FUNCTION_BLOCK FB_GripperAction
VAR_INPUT
    bExecute       : BOOL;
    eCommand       : E_GripperCommand;
    bCancel        : BOOL;
    bAllowCloseTargetWithoutGrip : BOOL := FALSE;
    tAcceptTimeout : TIME := GVL_ProcessConfig.stGripper.tAcceptTimeout;
    tResultTimeout : TIME := GVL_ProcessConfig.stGripper.tResultTimeout;
END_VAR
VAR_IN_OUT
    ioGripper : ST_GripperInterface;
END_VAR
VAR_OUTPUT
    bBusy       : BOOL;
    bDone       : BOOL;
    bCloseTargetReachedWithoutGrip : BOOL;
    bError      : BOOL;
    udErrorCode : UDINT;
    udiActionId : UDINT;
    eStep       : E_GripperActionStep := E_GripperActionStep.Idle;
END_VAR
VAR
    bInitialized     : BOOL;
    bExecutePrevious : BOOL;
    eActiveCommand   : E_GripperCommand;
    bActiveAllowCloseTargetWithoutGrip : BOOL;
    fbAcceptTimeout  : TON;
    fbResultTimeout  : TON;
END_VAR

// 自动动作只写AutoCmd；底层Cmd由FB_GripperManager唯一生成。
IF NOT bInitialized THEN
    bExecutePrevious := bExecute;
    bInitialized := TRUE;
END_IF;

// 取消/释放只撤销特殊完成授权，不改变既有Stop/Fault链。
IF bCancel OR NOT bExecute THEN
    ioGripper.AutoCmd.bAllowCloseTargetWithoutGrip := FALSE;
    bActiveAllowCloseTargetWithoutGrip := FALSE;
    bCloseTargetReachedWithoutGrip := FALSE;
END_IF;

fbAcceptTimeout(
    IN := (eStep = E_GripperActionStep.WaitAccepted),
    PT := tAcceptTimeout
);
fbResultTimeout(
    IN := (eStep = E_GripperActionStep.WaitCompleted),
    PT := tResultTimeout
);

IF ((eStep = E_GripperActionStep.WaitAccepted)
    OR (eStep = E_GripperActionStep.WaitCompleted))
    AND (bCancel OR NOT bExecute) THEN
    bBusy := FALSE;
    bDone := FALSE;
    bError := TRUE;
    udErrorCode := TO_UDINT(E_GripperErrorCode.ActionCancelled);
    eStep := E_GripperActionStep.Error;
    bExecutePrevious := bExecute;
    RETURN;
END_IF;

CASE eStep OF
    E_GripperActionStep.Idle:
        bBusy := FALSE;
        bDone := FALSE;
        bCloseTargetReachedWithoutGrip := FALSE;
        bActiveAllowCloseTargetWithoutGrip := FALSE;
        bError := FALSE;
        udErrorCode := TO_UDINT(E_GripperErrorCode.None);

        IF bExecute AND NOT bExecutePrevious AND NOT bCancel THEN
            IF (eCommand <> E_GripperCommand.Close)
                AND (eCommand <> E_GripperCommand.Open)
                AND (eCommand <> E_GripperCommand.Enable) THEN
                bError := TRUE;
                udErrorCode := TO_UDINT(E_GripperErrorCode.ActionInvalidCommand);
                eStep := E_GripperActionStep.Error;
            ELSE
                eActiveCommand := eCommand;
                bActiveAllowCloseTargetWithoutGrip :=
                    bAllowCloseTargetWithoutGrip
                    AND (eActiveCommand = E_GripperCommand.Close);
                ioGripper.AutoCmd.bAllowCloseTargetWithoutGrip :=
                    bActiveAllowCloseTargetWithoutGrip;
                ioGripper.AutoCmd.eCommand := eActiveCommand;
                IF ioGripper.AutoCmd.udiRequestId = 16#FFFFFFFF THEN
                    ioGripper.AutoCmd.udiRequestId := 1;
                ELSE
                    ioGripper.AutoCmd.udiRequestId :=
                        ioGripper.AutoCmd.udiRequestId + 1;
                END_IF;
                udiActionId := ioGripper.AutoCmd.udiRequestId;
                bBusy := TRUE;
                eStep := E_GripperActionStep.WaitAccepted;
            END_IF;
        END_IF;

    E_GripperActionStep.WaitAccepted:
        IF ioGripper.AutoFeedback.udiRejectedId = udiActionId THEN
            bBusy := FALSE;
            bError := TRUE;
            udErrorCode := ioGripper.AutoFeedback.udErrorCode;
            IF udErrorCode = TO_UDINT(E_GripperErrorCode.None) THEN
                udErrorCode := TO_UDINT(E_GripperErrorCode.ActionResultInvalid);
            END_IF;
            eStep := E_GripperActionStep.Error;
        ELSIF ioGripper.AutoFeedback.udiFailedId = udiActionId THEN
            bBusy := FALSE;
            bError := TRUE;
            udErrorCode := ioGripper.AutoFeedback.udErrorCode;
            IF udErrorCode = TO_UDINT(E_GripperErrorCode.None) THEN
                udErrorCode := TO_UDINT(E_GripperErrorCode.ActionResultInvalid);
            END_IF;
            eStep := E_GripperActionStep.Error;
        ELSIF ioGripper.AutoFeedback.udiAcceptedId = udiActionId THEN
            eStep := E_GripperActionStep.WaitCompleted;
        ELSIF fbAcceptTimeout.Q THEN
            bBusy := FALSE;
            bError := TRUE;
            udErrorCode := TO_UDINT(E_GripperErrorCode.ActionAcceptTimeout);
            eStep := E_GripperActionStep.Error;
        END_IF;

    E_GripperActionStep.WaitCompleted:
        IF ioGripper.AutoFeedback.udiFailedId = udiActionId THEN
            bBusy := FALSE;
            bError := TRUE;
            udErrorCode := ioGripper.AutoFeedback.udErrorCode;
            IF udErrorCode = TO_UDINT(E_GripperErrorCode.None) THEN
                udErrorCode := TO_UDINT(E_GripperErrorCode.ActionResultInvalid);
            END_IF;
            eStep := E_GripperActionStep.Error;
        ELSIF ioGripper.AutoFeedback.udiCompletedId = udiActionId THEN
            IF ioGripper.State.bHealthy
                AND ((eActiveCommand <> E_GripperCommand.Enable)
                    OR (ioGripper.AutoFeedback.udErrorCode = TO_UDINT(E_GripperErrorCode.None)))
                AND ((eActiveCommand = E_GripperCommand.Enable)
                    OR NOT ioGripper.AutoFeedback.bCloseTargetReachedWithoutGrip
                    OR bActiveAllowCloseTargetWithoutGrip) THEN
                bBusy := FALSE;
                bCloseTargetReachedWithoutGrip :=
                    ioGripper.AutoFeedback.bCloseTargetReachedWithoutGrip;
                bDone := TRUE;
                eStep := E_GripperActionStep.Done;
            ELSE
                bBusy := FALSE;
                bError := TRUE;
                udErrorCode := TO_UDINT(E_GripperErrorCode.ActionResultInvalid);
                eStep := E_GripperActionStep.Error;
            END_IF;
        ELSIF fbResultTimeout.Q THEN
            bBusy := FALSE;
            bError := TRUE;
            udErrorCode := TO_UDINT(E_GripperErrorCode.ActionResultTimeout);
            eStep := E_GripperActionStep.Error;
        END_IF;

    E_GripperActionStep.Done:
        bBusy := FALSE;
        IF NOT bExecute THEN
            bDone := FALSE;
            eStep := E_GripperActionStep.Idle;
        ELSIF NOT ioGripper.State.bHealthy
            OR (ioGripper.AutoFeedback.udiCompletedId <> udiActionId) THEN
            bDone := FALSE;
            bError := TRUE;
            udErrorCode := TO_UDINT(E_GripperErrorCode.ActionResultInvalid);
            eStep := E_GripperActionStep.Error;
        END_IF;

    E_GripperActionStep.Error:
        bBusy := FALSE;
        bError := TRUE;
        bCloseTargetReachedWithoutGrip := FALSE;
        bActiveAllowCloseTargetWithoutGrip := FALSE;
        ioGripper.AutoCmd.bAllowCloseTargetWithoutGrip := FALSE;
        IF NOT bExecute THEN
            bError := FALSE;
            eStep := E_GripperActionStep.Idle;
        END_IF;
END_CASE;

IF bError THEN
    bCloseTargetReachedWithoutGrip := FALSE;
    bActiveAllowCloseTargetWithoutGrip := FALSE;
    ioGripper.AutoCmd.bAllowCloseTargetWithoutGrip := FALSE;
END_IF;

bExecutePrevious := bExecute;

END_FUNCTION_BLOCK

(* stored: Version 1.1.0.1, ProductVersion 3.1.4026.20
   POU FB_GripperAction: Id {c2ce23f6-bc7d-437a-91da-351ba974928b}, SpecialFunc None *)
